FUNCTION_BLOCK FB_ScorerHeight
VAR_INPUT

	EN					: BOOL;
	autoManual			: BOOL;

	manualIncrement		: BOOL;
	manualDecrement		: BOOL;
	circuitBreaker		: BOOL;
	limitMax			: BOOL;
	limitMin			: BOOL;
	scorerHeightPositionSensor	: WORD;
	fluteType			: STRING;
	scorerHeightArr		: ARRAY [1..5] OF REAL;	(*Scorer height setpoint*)


END_VAR
VAR_OUTPUT

	ENO						: BOOL;
	error					: BOOL;
	positionIncrement		: BOOL;
	positionDecrement		: BOOL;
	scorerHeightMM			: REAL;				(*Scorer height position actual value in milimiters*)
	scorerHeightDifMM		: REAL;	(*Diference btween setpoint and actual value*)

END_VAR
VAR
END_VAR


(*==============================================================================================================================
CPNTeck - Automação industrial
(c)Copyright 2023 All Rights Reserved
_______________________________________________________________________________________________________________________________
Library: N/A 
Tested with: CX5140
Engineering: Twincat 2
Restrictions: -
Requirements: N/A
Functionality: This function is used control the scorer height positioning
Support: fabio@cpnteck.com.br
Note: Parameter comments are only available in language 'English (United States)'
_______________________________________________________________________________________________________________________________
Change log table:

Version  		| Date        			| Expert in charge  	| Changes applied
01.00.01		| 29.03.2023  		| Fabio Campion            | First released version



===============================================================================================================================*)

ACT_IncrementDecrement();
ACT_ScorerHeightSensor();

ACTION ACT_IncrementDecrement:
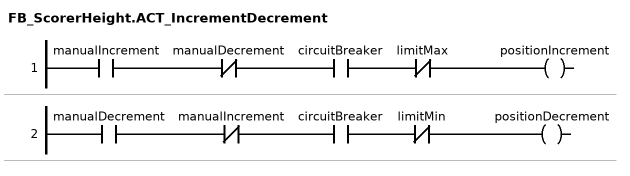
// NETWORK 1
positionIncrement := manualIncrement AND NOT manualDecrement AND circuitBreaker AND NOT limitMax;

// NETWORK 2
positionDecrement := manualDecrement AND NOT manualIncrement AND circuitBreaker AND NOT limitMin;
END_ACTION

ACTION ACT_ScorerHeightSensor:


scorerHeightMM := SCALE_R(
	X:= scorerHeightPositionSensor, 
	I_LO:= 7120, 
	I_HI:= 23880, 
	O_LO:= 3, 
	O_HI:= 0);
END_ACTION

END_FUNCTION_BLOCK

(* stored: Version 1.1.0.1
   POU FB_ScorerHeight: Id {02a244b8-a79b-4e14-9827-78669c61d068}, SpecialFunc None
   Action ACT_IncrementDecrement: Id {965c1db3-1274-4358-b1ea-f89656f3acfd}
   Action ACT_ScorerHeightSensor: Id {7cf5766f-d4bf-4c6a-9f9d-64ee30a393cc} *)
